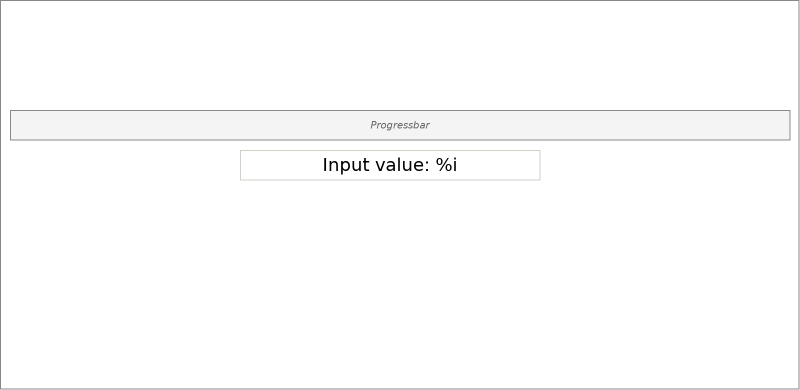
VISUALIZATION VisuAnlogInputControl  // 800x390
    Rectangle (0,0 800x390)
    Progressbar (10,110 780x30), variable: GVL_DevManual.fbManualControler.pDevAnalogInput^.fValue
    Textfield (240,150 300x30), "Input value: %i", text variable: GVL_DevManual.fbManualControler.pDevAnalogInput^.fValue
END_VISUALIZATION

(* stored: Version 1.1.0.1, ProductVersion 3.1.4024.5
   Visu VisuAnlogInputControl: Id {05161f7c-ba6d-4f2f-9bcb-245dad7521da} *)
